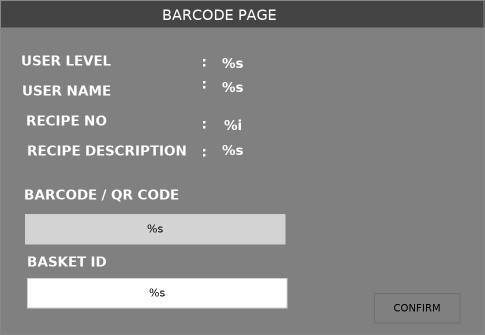
VISUALIZATION Popup_Barcode  // 485x335
    Rectangle (0,0 485x335)
    Rectangle (0,0 485x27)
    Label (159,3 146x24), "BARCODE PAGE"
    Rectangle (219,79 169x17), "%s", text variable: fbHmiTF1800_UserlevelManagement.dsHmiUserReg.ARwsUserGroupName[iLoginNameId]
    Rectangle (219,55 169x17), "%s", text variable: fbHmiTF1800_UserlevelManagement.dsHmiUserReg.ARsLoginName[iLoginNameId]
    Label (18,49 180x24), "USER LEVEL"
    Label (200,57 10x10), ":"
    Label (19,79 179x24), "USER NAME"
    Label (200,79 10x10), ":"
    Label (23,109 177x24), "RECIPE NO"
    Label (200,119 10x10), ":"
    Label (23,139 167x24), "RECIPE DESCRIPTION"
    Label (200,147 10x10), ":"
    Rectangle (221,117 62x17), "%i", text variable: HMI_Function.iRecipeNoFeed
    Rectangle (219,142 169x17), "%s", text variable: ARsProductRecipeDescription[HMI_Function.iRecipeNoFeed]
    Textfield (25,214 260x30), "%s", text variable: sBarcodeScannerReceivedCmd
    Label (21,183 261x24), "BARCODE / QR CODE"
    Button (374,293 86x30), "CONFIRM", colour toggle: bBarcodeConfirm
        tap bBarcodeConfirm
        OnMouseClick: change screen: AutoMain_Page
    Label (24,250 258x24), "BASKET ID"
    Textfield (27,278 260x30), "%s", text variable: sBasketNo
        OnMouseDown: write the text variable via VisuDialogs.Keypad
END_VISUALIZATION

(* stored: Version 1.1.0.1, ProductVersion 3.1.4024.12
   Visu Popup_Barcode: Id {bbaa8915-e670-435b-8acc-808737343505} *)
